// TIA Portal V20 export
DATA_BLOCK "DB_ConveyorParameters"   // DB27
// stored: Access Published, MemoryReserve 100, Namespace LineD1
   VAR
      Line : Struct
         D1 : Struct
            Conveyor : Array[_.minD1.._.maxD1] of "LineD1.ConveyorParameters";
         END_STRUCT;
      END_STRUCT;
   END_VAR
BEGIN
END_DATA_BLOCK
